// TwinCAT 3 PLC project PLC1
// ProgramVersion: 3.1.4023.0
// libraries:
//   Tc2_ModbusSrv, * (Beckhoff Automation GmbH)
//   Tc2_Standard, * (Beckhoff Automation GmbH)
//   Tc2_System, * (Beckhoff Automation GmbH)
//   Tc3_Module, * (Beckhoff Automation GmbH)
// project tree:
//   / PlcTask.TcTTO
//   POUs/Basic_MGS/ FB_Blinking.TcPOU
//   POUs/ ClassDiagram.TcCD (not stored), PRG_MAIN.TcPOU
//   POUs/FactoryIO_MGS/BasicDep/ FB_Bool_To_Word.TcPOU (not stored), FB_Word_To_Bool.TcPOU (not stored)
//   POUs/FactoryIO_MGS/ FB_Exercice1.TcPOU, FB_FactoryIO_ModbusTCP_Read.TcPOU, FB_FactoryIO_ModbusTCP_Write.TcPOU, GVL_FactoryIO.TcGVL, PRG_FactoryIO_ModbusTCP_Read.TcPOU, PRG_FactoryIO_ModbusTCP_Write.TcPOU
//   POUs/FactoryIO_MGS/Old/ PRG_FactoryIO_ModbusTCP_old.TcPOU
//   POUs/FactoryIO_WebSample/ F_FactoryIO_Read_InputRegs.TcPOU, F_FactoryIO_Read_Inputs.TcPOU (not stored), F_FactoryIO_WriteRegs.TcPOU, F_FactoryIO_Write_Coils.TcPOU, GVL_FactoryIO_WebSample.TcGVL
// real-time tasks:
//   TASK PlcTask: cycle T#50000us, priority 20, ADS port 350

CONFIGURATION PLC1
    RESOURCE PLC ON TwinCAT3
        TASK PlcTask(INTERVAL := T#50000us, PRIORITY := 20);
        PROGRAM PRG_FactoryIO_ModbusTCP_Read WITH PlcTask : PRG_FactoryIO_ModbusTCP_Read;
        PROGRAM PRG_MAIN WITH PlcTask : PRG_MAIN;
        PROGRAM PRG_FactoryIO_ModbusTCP_Write WITH PlcTask : PRG_FactoryIO_ModbusTCP_Write;
    END_RESOURCE
END_CONFIGURATION

// ---- POUs/FactoryIO_MGS/GVL_FactoryIO.TcGVL
VAR_GLOBAL
	

	// FIO (FactoryIO)
	FIO_Input1: ARRAY [0..15] OF BOOL;
	FIO_Input2: ARRAY [0..15] OF BOOL;
	FIO_InputReg: ARRAY [0..7] OF INT;
	FIO_Output1: ARRAY [0..15] OF BOOL;
	FIO_Output2: ARRAY [0..15] OF BOOL;
	FIO_OutputReg: ARRAY [0..7] OF INT;
	
	// Exercice 1 (penser à modifier aussi dans mapping
	// Entrées
	E_BoutonMarche: BOOL;
	E_Capteur: BOOL;
	E_BoutonAvancer: BOOL;
	// Sorties
	S_VoyantMarche: BOOL;
	S_Convoyeur: BOOL;
	S_VoyantAvancer: BOOL;
	
END_VAR

// ---- POUs/FactoryIO_WebSample/GVL_FactoryIO_WebSample.TcGVL
VAR_GLOBAL
//	GAB_FactoryIO_Inputs : ARRAY [0..1] OF WORD;
//	GAB_FactoryIO_InputRegs : ARRAY [0..7] OF INT;
//	GAB_FactoryIO_Outputs : ARRAY [0..1] OF WORD;
//	GAB_FactoryIO_OutputsRegs : ARRAY [0..7] OF INT;
END_VAR

// ---- POUs/FactoryIO_MGS/PRG_FactoryIO_ModbusTCP_Read.TcPOU
PROGRAM PRG_FactoryIO_ModbusTCP_Read
// Dépendance Tc2_ModbusSrv (TF6250-Modbus-TCP)
// FB_Bool_To_Word + FB_Word_To_Bool
VAR
	fb_FactoryIO_ModbusTCP_Read : FB_FactoryIO_ModbusTCP_Read;
END_VAR

// READ ModbusTCP FactoryIO
fb_FactoryIO_ModbusTCP_Read();
// Call method
fb_FactoryIO_ModbusTCP_Read.ReadInput();
fb_FactoryIO_ModbusTCP_Read.ReadInputRegister();
FIO_InputReg := fb_FactoryIO_ModbusTCP_Read.InputReg;
FIO_Input1 := fb_FactoryIO_ModbusTCP_Read.bInput1;
FIO_Input2 := fb_FactoryIO_ModbusTCP_Read.bInput2;
fb_FactoryIO_ModbusTCP_Read.MappingInput();

END_PROGRAM

// ---- POUs/FactoryIO_MGS/FB_FactoryIO_ModbusTCP_Read.TcPOU
FUNCTION_BLOCK PUBLIC FB_FactoryIO_ModbusTCP_Read
VAR_INPUT
	// **** Configuration en fonction de la configuration FactoryIO
	sIPAddr : STRING[15]:='127.0.0.1'; // '127.0.0.1'
	nTCPPort : UINT:=505; // 505
	nUnitID : BYTE:=255; // 255	
END_VAR

VAR_OUTPUT
	bBusy: BOOL;
	bError: BOOL;
	// *** Configuration des array en fonction de la configuration FactoryIO
	InputReg : ARRAY [0..7] OF INT; // ex. input register 8 [0..7] pour les mesures analogiques
	// Inputs traités
	bInput1 : ARRAY [0..15] OF BOOL;
	bInput2 : ARRAY [0..15] OF BOOL;
	
END_VAR
	
VAR
	// Instances
	fb_MBReadInputs : FB_MBReadInputs; // Instance de la fonction FB_MBReadInputs de la lib Tc2_ModbusSrv
	fb_MBReadInputRegs : FB_MBReadInputRegs;
	
	fb_Word_To_Bool : FB_Word_To_Bool; // Instance commune
	fb_Bool_To_Word: FB_Bool_To_Word ; // Instance commune
	
	// *** Configuration des array en fonction de la configuration FactoryIO
	Input : ARRAY [0..1] OF WORD; // ex. input digital 16 [0..0] /  input digital 32 [0..1]
	
	// Busy Error interne à la fonciton
	bBusyInput: ARRAY [1..2] OF BOOL;
	bErrorInput: ARRAY [1..2] OF BOOL;

END_VAR

// Traitement des bool représentant les inputs
fb_Word_To_Bool(inWord := Input[0],
				outArrayOfBool => bInput1);
fb_Word_To_Bool(inWord := Input[1],
				outArrayOfBool => bInput2);
				
			

// Busy si au moins 1 busy
IF bBusyInput[1] OR bBusyInput[2] THEN
	bBusy := 1;
ELSE
	bBusy := 0;
END_IF

// Error si au moins 1 busy
IF bErrorInput[1] OR bErrorInput[2] THEN
	bError := 1;
ELSE
	bError := 0;
END_IF

METHOD MappingInput
VAR_INPUT
END_VAR
// Exercice 1
E_BoutonMarche := FIO_Input1[0];
E_Capteur := FIO_Input1[1];
E_BoutonAvancer := FIO_Input1[2];
END_METHOD

METHOD PUBLIC ReadInput
fb_MBReadInputs(
	sIPAddr := sIPAddr,
	nTCPPort := nTCPPort,
	nUnitID := nUnitID,
	nQuantity := SIZEOF(Input)*8, // Nombre de bits à lire SIZEOF(nb byte * bits dans 1 byte)
	nMBAddr := 0,
	cbLength := SIZEOF(Input),
	pDestAddr := ADR(Input),
	bExecute := TRUE,
	tTimeout := T#1S,
	bBusy => bBusyInput[1],
	bError => bErrorInput[1],
	nErrId => ,
	cbRead => ,
 );
fb_MBReadInputs(bExecute := FALSE);
END_METHOD

METHOD PUBLIC ReadInputRegister
fb_MBReadInputRegs(
	sIPAddr := sIPAddr,
	nTCPPort := nTCPPort,
	nUnitID := nUnitID,
	nQuantity := SIZEOF(InputReg)/2,
	nMBAddr := 0,
	cbLength := SIZEOF(InputReg),
	pDestAddr := ADR(InputReg),
	bExecute := TRUE,
	tTimeout := T#1S,
	bBusy => bBusyInput[2],
	bError => bErrorInput[2],
	nErrId => ,
	cbRead => ,
 );
fb_MBReadInputRegs(bExecute := FALSE);
END_METHOD

END_FUNCTION_BLOCK

// ---- POUs/PRG_MAIN.TcPOU
PROGRAM PRG_MAIN
VAR
	fb_Blinking : ARRAY [0..1] OF FB_Blinking;
	fb_Exercice1: FB_Exercice1;
END_VAR


fb_Exercice1();

//fb_Blinking[0](Enable:=1 , PT_OFF:= , PT_ON:= , Output=>FIO_Output1[0]);
////fb_Blinking[1](Enable:=1 , PT_OFF:=T#1S, PT_ON:=T#3S, Output=>FIO_Output1[1]);

//IF FIO_I_Capteur THEN
//	FIO_O_Convoyeur := 1;
//ELSE
//	FIO_O_Convoyeur := 0;
//END_IF

END_PROGRAM

// ---- POUs/Basic_MGS/FB_Blinking.TcPOU
FUNCTION_BLOCK PUBLIC FB_Blinking
VAR_INPUT
	Enable: BOOL;
	PT_OFF: TIME :=T#0.7S;
	PT_ON: TIME := T#1S;
END_VAR
VAR_OUTPUT
	Output: BOOL;
END_VAR
VAR
	TON1_OFF: TON;
	TON2_ON: TON;
END_VAR

	
IF Enable THEN
	TON1_OFF(IN:= , PT:=PT_OFF , Q=> , ET=> );
	TON2_ON(IN:= , PT:=PT_ON , Q=> , ET=> );
	
	TON1_OFF.IN := NOT TON2_ON.Q;
	TON2_ON.IN := TON1_OFF.Q;
	
	IF TON1_OFF.Q THEN
		Output := 1;
	ELSE
		Output := 0;
	END_IF	
END_IF

END_FUNCTION_BLOCK

// ---- POUs/FactoryIO_MGS/FB_Exercice1.TcPOU
FUNCTION_BLOCK FB_Exercice1
VAR_INPUT
END_VAR
VAR_OUTPUT
END_VAR
VAR
	fb_Blinking : ARRAY [0..1] OF FB_Blinking;
END_VAR

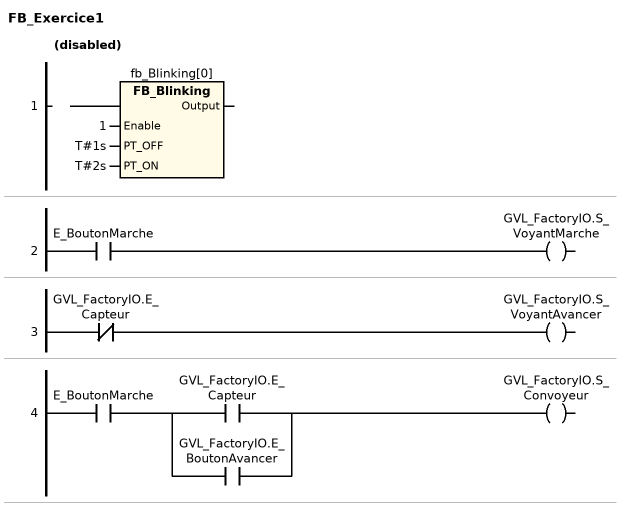
// NETWORK 1 (disabled)
// fb_Blinking[0](Enable := 1, PT_OFF := T#1s, PT_ON := T#2s); // FB_Blinking

// NETWORK 2
GVL_FactoryIO.S_VoyantMarche := E_BoutonMarche;

// NETWORK 3
GVL_FactoryIO.S_VoyantAvancer := NOT GVL_FactoryIO.E_Capteur;

// NETWORK 4
GVL_FactoryIO.S_Convoyeur := E_BoutonMarche AND (GVL_FactoryIO.E_Capteur OR GVL_FactoryIO.E_BoutonAvancer);

END_FUNCTION_BLOCK

// ---- POUs/FactoryIO_MGS/PRG_FactoryIO_ModbusTCP_Write.TcPOU
PROGRAM PRG_FactoryIO_ModbusTCP_Write
// Dépendance Tc2_ModbusSrv (TF6250-Modbus-TCP)
// FB_Bool_To_Word + FB_Word_To_Bool
VAR
	fb_FactoryIO_ModbusTCP_Write : FB_FactoryIO_ModbusTCP_Write;
END_VAR

fb_FactoryIO_ModbusTCP_Write.MappingOutput();
// WRITE ModbusTCP FactoryIO
fb_FactoryIO_ModbusTCP_Write(OutputReg := FIO_OutputReg, bOutput1 := FIO_Output1, bOutput2 := FIO_Output2);
// Call method
fb_FactoryIO_ModbusTCP_Write.WriteOutput();
fb_FactoryIO_ModbusTCP_Write.WriteOutputRegister();

END_PROGRAM

// ---- POUs/FactoryIO_MGS/FB_FactoryIO_ModbusTCP_Write.TcPOU
FUNCTION_BLOCK PUBLIC FB_FactoryIO_ModbusTCP_Write
VAR_INPUT
	// **** Configuration en fonction de la configuration FactoryIO
	sIPAddr : STRING[15]:='127.0.0.1'; // '127.0.0.1'
	nTCPPort : UINT:=505; // 505
	nUnitID : BYTE:=255; // 255
	
	// **** Configuration des array en fonction de la configuration FactoryIO
	OutputReg : ARRAY [0..7] OF INT;
	// Outpus traités
	bOutput1 : ARRAY [0..15] OF BOOL;
	bOutput2 : ARRAY [0..15] OF BOOL;
	
END_VAR

VAR_OUTPUT
	bBusy: BOOL;
	bError: BOOL;
	
END_VAR
	
VAR
	// Instances
	fb_MBWriteCoils : FB_MBWriteCoils; // Instance de la fonction FB_MBReadInputs de la lib Tc2_ModbusSrv
	fb_MBWriteRegs : FB_MBWriteRegs ;
	
	fb_Word_To_Bool : FB_Word_To_Bool; // Instance commune
	fb_Bool_To_Word: FB_Bool_To_Word ; // Instance commune
	
	// **** Configuration des array en fonction de la configuration FactoryIO
	Output : ARRAY [0..1] OF WORD;
	
	// Busy Error interne à la fonciton
	bBusyInput: ARRAY [1..2] OF BOOL;
	bErrorInput: ARRAY [1..2] OF BOOL;

END_VAR

// Traitement des bool représentant les outputs
fb_Bool_To_Word(inArrayOfBool := bOutput1,
				outWord => Output[0]);
fb_Bool_To_Word(inArrayOfBool := bOutput2,
				outWord => Output[1]);	
				

// Busy si au moins 1 busy
IF bBusyInput[1] OR bBusyInput[2] THEN
	bBusy := 1;
ELSE
	bBusy := 0;
END_IF

// Error si au moins 1 busy
IF bErrorInput[1] OR bErrorInput[2] THEN
	bError := 1;
ELSE
	bError := 0;
END_IF

METHOD MappingOutput
VAR_INPUT
END_VAR
// Exercice 1
FIO_Output1[0] := S_VoyantMarche;
FIO_Output1[1] := S_Convoyeur;
FIO_Output1[2] := S_VoyantAvancer;
END_METHOD

METHOD PUBLIC WriteOutput
fb_MBWriteCoils(
	sIPAddr := sIPAddr,
	nTCPPort := nTCPPort,
	nUnitID := nUnitID,
	nQuantity := SIZEOF(Output)*8,
	nMBAddr := 0,
	cbLength := SIZEOF(Output),
	pSrcAddr := ADR(Output),
	bExecute := TRUE,
	tTimeout := T#1S,
	bBusy => bBusyInput[1],
	bError => bErrorInput[1],
	nErrId => ,
 );
fb_MBWriteCoils(bExecute := FALSE);
END_METHOD

METHOD PUBLIC WriteOutputRegister
fb_MBWriteRegs(
	sIPAddr := sIPAddr,
	nTCPPort := nTCPPort,
	nUnitID := nUnitID,
	nQuantity := SIZEOF(OutputReg)/2,
	nMBAddr := 0,
	cbLength := SIZEOF(OutputReg),
	pSrcAddr := ADR(OutputReg),
	bExecute := TRUE,
	tTimeout := T#1S,
	bBusy => bBusyInput[2],
	bError => bErrorInput[2],
	nErrId => ,
 );
fb_MBWriteRegs(bExecute := FALSE);
END_METHOD

END_FUNCTION_BLOCK

// ---- POUs/FactoryIO_MGS/Old/PRG_FactoryIO_ModbusTCP_old.TcPOU
PROGRAM PRG_FactoryIO_ModbusTCP_old
// Dépendance Tc2_ModbusSrv (TF6250-Modbus-TCP)
// FB_Bool_To_Word + FB_Word_To_Bool
VAR
	fb_FactoryIO_ModbusTCP : FB_FactoryIO_ModbusTCP_Read;
END_VAR

FIO_Input1 := fb_FactoryIO_ModbusTCP.bInput1;
FIO_Input2 := fb_FactoryIO_ModbusTCP.bInput;
FIO_InputReg := fb_FactoryIO_ModbusTCP.InputReg;
fb_FactoryIO_ModbusTCP.Write_Output();
fb_FactoryIO_ModbusTCP.Write_OutputRegister();
// Call method
fb_FactoryIO_ModbusTCP.Input();
// READ WRITE ModbusTCP FactoryIO
fb_FactoryIO_ModbusTCP(
    sIPAddr := '127.0.0.1',
    nTCPPort := 505,
    nUnitID := 255,
    OutputReg := FIO_OutputReg,
    bOutput1 := FIO_Output1,
    bOutput2 := FIO_Output2); // FB_FactoryIO_ModbusTCP_Read
fb_FactoryIO_ModbusTCP.ReadInputRegister();

END_PROGRAM

// ---- POUs/FactoryIO_WebSample/F_FactoryIO_Read_InputRegs.TcPOU
PROGRAM F_FactoryIO_Read_InputRegs
VAR;
	LFB_MBReadInputRegs 	: FB_MBReadInputRegs;
	bBusy: BOOL;
	bError: BOOL;
END_VAR

LFB_MBReadInputRegs(
	sIPAddr := '127.0.0.1',
	nTCPPort := 505,
	nUnitID := 255,
	nQuantity := 8, // Nombre de registres à lire
	nMBAddr := 0,
	cbLength := SIZEOF(GAB_FactoryIO_InputRegs),
	pDestAddr := ADR(GAB_FactoryIO_InputRegs),
	bExecute := TRUE,
	tTimeout := T#1S,
	bBusy => bBusy,
	bError => bError,
	nErrId => ,
	cbRead => ,
 );
 
 
 
 
LFB_MBReadInputRegs(bExecute := FALSE);

END_PROGRAM

// ---- POUs/FactoryIO_WebSample/F_FactoryIO_WriteRegs.TcPOU
PROGRAM F_FactoryIO_WriteRegs
VAR
	LFB_MBWriteRegs  	: FB_MBWriteRegs ;
	bBusy: BOOL;
	bError: BOOL;

END_VAR

LFB_MBWriteRegs(
	sIPAddr := '127.0.0.1',
	nTCPPort := 505,
	nUnitID := 255,
	nQuantity := 8,
	nMBAddr := 0,
	cbLength := SIZEOF(GAB_FactoryIO_OutputsRegs),
	pSrcAddr:= ADR(GAB_FactoryIO_OutputsRegs), 
	bExecute := TRUE,
	tTimeout := T#1S,
	bBusy=> bBusy, 
	bError=> bError, 
	nErrId=>
);
LFB_MBWriteRegs(bExecute := FALSE);

END_PROGRAM

// ---- POUs/FactoryIO_WebSample/F_FactoryIO_Write_Coils.TcPOU
PROGRAM F_FactoryIO_Write_Coils
VAR
	LFB_MBWriteCoils 	: FB_MBWriteCoils;
	bBusy: BOOL;
	bError: BOOL;

END_VAR

LFB_MBWriteCoils(
	sIPAddr := '127.0.0.1',
	nTCPPort := 505,
	nUnitID := 255,
	nQuantity := 16,
	nMBAddr := 0,
	cbLength := SIZEOF(GAB_FactoryIO_Outputs),
	pSrcAddr:= ADR(GAB_FactoryIO_Outputs), 
	bExecute := TRUE,
	tTimeout := T#1S,
	bBusy=> bBusy, 
	bError=> bError, 
	nErrId=>
);
LFB_MBWriteCoils(bExecute := FALSE);

END_PROGRAM
